// TwinCAT 3 PLC project XtesSxrPlc
// ProgramVersion: 3.1.4022.3
// libraries:
//   L2Si Vacuum Library, * (SLAC)
//   Tc2_Standard, * (Beckhoff Automation GmbH)
//   Tc2_System, * (Beckhoff Automation GmbH)
//   Tc3_Module, * (Beckhoff Automation GmbH)
// project tree:
//   GVLs/ GVL_DEVICES.TcGVL, GVL_VARIABLES.TcGVL
//   / PlcTask.TcTTO
//   POUs/ MAIN.TcPOU, PRG_PROTOTYPE.TcPOU
// real-time tasks:
//   TASK PlcTask: cycle T#10ms, priority 20, ADS port 350
// I/O:
//   DEVICE =+-AuxPS1-CPU/EtherCAT1, AmsNetId 10.0.1.22.2.1
//     =+-AuxPS1 [EK1100 EtherCAT Coupler (2A E-Bus)]
//       =+-DO1 [EL2794 4Ch. Dig. Output 24V AC/DC, 2A, short-circuit-proof]
//       =+-DI1 [EL1004 4Ch. Dig. Input 24V, 3ms]
//     =+-A1 [EP2338-0002 8 Ch. Dig. Input/Output 24V, 0,5A, M12]
//     =+-A2 [EP3174-0002 4Ch. Ana. Input +/-10V, 0-10V, 0/4-20mA configurable]
//     =+-A3 [EP2624-0002 4Ch. Relay Output, NO (125V AC / 30V DC)]
// variable links:
//   XtesSxrPlc/XtesSxrPlc Instance <-> =+-AuxPS1-CPU/EtherCAT1/=+-A1
//     PlcTask Inputs/GVL_DEVICES.MR1K4_VGC_1.i_xClsLS <-> Channel 4/Input
//     PlcTask Inputs/GVL_DEVICES.MR1K4_VGC_1.i_xOpnLS <-> Channel 3/Input
//     PlcTask Inputs/GVL_DEVICES.TV2K4_VGC_1.i_xClsLS <-> Channel 8/Input
//     PlcTask Inputs/GVL_DEVICES.TV2K4_VGC_1.i_xOpnLS <-> Channel 7/Input
//     PlcTask Outputs/GVL_DEVICES.MR1K4_VGC_1.q_xOPN_DO <-> Channel 9/Output
//     PlcTask Outputs/GVL_DEVICES.TV2K4_VGC_1.q_xOPN_DO <-> Channel 13/Output
//   XtesSxrPlc/XtesSxrPlc Instance <-> =+-AuxPS1-CPU/EtherCAT1/=+-A2
//     PlcTask Inputs/GVL_DEVICES.TV2K4_GCC_1.i_iPRESS_R <-> AI Standard Channel 1/Value
//     PlcTask Inputs/GVL_DEVICES.TV2K4_GPI_1.i_iPRESS_R <-> AI Standard Channel 4/Value
//   XtesSxrPlc/XtesSxrPlc Instance <-> =+-AuxPS1-CPU/EtherCAT1/=+-A3
//     PlcTask Outputs/GVL_DEVICES.TV2K4_GCC_1.q_xHV_DIS <-> Channel 1/Output
//   XtesSxrPlc/XtesSxrPlc Instance <-> =+-AuxPS1-CPU/EtherCAT1/=+-AuxPS1/=+-DI1
//     PlcTask Inputs/GVL_DEVICES.TV2KO_PIP_1.i_xSP_DI <-> Channel 4/Input
//   XtesSxrPlc/XtesSxrPlc Instance <-> =+-AuxPS1-CPU/EtherCAT1/=+-AuxPS1/=+-DO1
//     PlcTask Outputs/GVL_DEVICES.TV2KO_PIP_1.q_xHVEna_DO <-> Channel 1/Output

CONFIGURATION XtesSxrPlc
    RESOURCE PLC ON TwinCAT3
        TASK PlcTask(INTERVAL := T#10ms, PRIORITY := 20);
        PROGRAM MAIN WITH PlcTask : MAIN;
    END_RESOURCE
END_CONFIGURATION

// ---- GVLs/GVL_DEVICES.TcGVL
VAR_GLOBAL
	
// gauges
	{attribute 'pytmc' := ' pv: MR2K3_GPI_1 '}
	MR2K3_GPI_1 : FB_MKS275;
	{attribute 'pytmc' := ' pv: TV2K4_GPI_1 '}
	TV2K4_GPI_1 : FB_MKS275;
	{attribute 'pytmc' := ' pv: MR1K4_GPI_1 '}
	MR1K4_GPI_1 : FB_MKS275;
	{attribute 'pytmc' := ' pv: MR2K3_GCC_1 '}
	MR2K3_GCC_1 : FB_MKS500;
	{attribute 'pytmc' := ' pv: TV2K4_GCC_1 '}
	TV2K4_GCC_1 : FB_MKS500;
	{attribute 'pytmc' := ' pv: MR1K4_GCC_1 '}
	MR1K4_GCC_1 : FB_MKS500;

//valves
	{attribute 'pytmc' := ' pv: TV2K4_VGC_1 '}
	TV2K4_VGC_1 : FB_VGC; // VV9S
	{attribute 'pytmc' := ' pv: MR1K4_VGC_1'}
	MR1K4_VGC_1 : FB_VGC; // VV10S
	
//pumps
	{attribute 'pytmc' := ' pv: TV2KO_PIP_1 '}
	TV2KO_PIP_1 : FB_PIP_Gamma;

END_VAR

// ---- GVLs/GVL_VARIABLES.TcGVL
VAR_GLOBAL
	{attribute 'pytmc' := 'pv: AT1L0:GAS:VAC:OVRDON'}
	xSystemOverrideMode : BOOL; (* Global system override for the prototype section*)
END_VAR

// ---- POUs/MAIN.TcPOU
PROGRAM MAIN
VAR
END_VAR

PRG_PROTOTYPE();

END_PROGRAM

// ---- POUs/PRG_PROTOTYPE.TcPOU
PROGRAM PRG_PROTOTYPE
VAR
END_VAR

//gauges
MR2K3_GPI_1(PG=>);
TV2K4_GPI_1(PG=>);
MR1K4_GPI_1(PG=>);

MR2K3_GCC_1(PG:=MR2K3_GPI_1.PG);
TV2K4_GCC_1(PG:=TV2K4_GPI_1.PG);
MR1K4_GCC_1(PG:=MR1K4_GPI_1.PG);

//valves
TV2K4_VGC_1(i_stUSG := MR2K3_GCC_1.IG, 
			i_stDSG:= TV2K4_GCC_1.IG, 
			i_xDis_DPIlk := TRUE, 
			i_xEPS_OK := TRUE, 
			i_xPMPS_OK := TRUE, 
			i_xExt_OK := TRUE, 
			i_xOverrideMode := xSystemOverrideMode);
			
MR1K4_VGC_1(i_stUSG := TV2K4_GCC_1.IG, 
			i_stDSG:= MR1K4_GCC_1.IG, 
			i_xDis_DPIlk := TRUE, 
			i_xEPS_OK := TRUE, 
			i_xPMPS_OK := TRUE, 
			i_xExt_OK := TRUE, 
			i_xOverrideMode := xSystemOverrideMode);
			
//pumps
TV2KO_PIP_1(i_stGauge:= TV2K4_GCC_1.IG);

END_PROGRAM
